% RSLogix 500 project STAR TO DELTA STARTER_BAK003.RSS, saved by version 8.30.00.16 %
PROJECT "UNTITLED"    % processor: Bul.1763 MicroLogix 1100 Series B %

PROGRAM FILES
  LAD 2   4 rungs

DATA FILES
  O0 OUTPUT  4 elements
  I1 INPUT  6 elements
  S2 STATUS  66 elements
  B3 BINARY  1 elements
  T4 TIMER  1 elements
  C5 COUNTER  1 elements
  R6 CONTROL  1 elements
  N7 INTEGER  1 elements
  F8 FLOAT  1 elements

LADDER 2
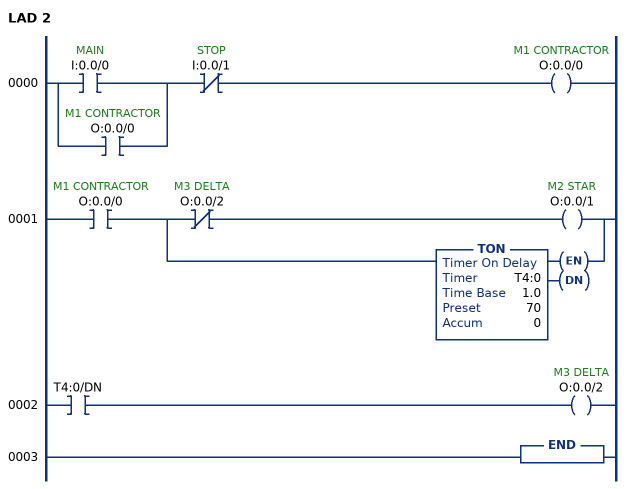
% Rung: 0 %  % edit flag set %
SOR BST XIC I:0.0/0 NXB XIC O:0.0/0 BND XIO I:0.0/1 OTE O:0.0/0 EOR
%   I:0.0/0  "MAIN" %
%   O:0.0/0  "M1 CONTRACTOR" %
%   I:0.0/1  "STOP" %
% Rung: 1 %  % edit flag set %
SOR XIC O:0.0/0 BST XIO O:0.0/2 OTE O:0.0/1 NXB TON T4:0 1.0 70 0 BND EOR
%   O:0.0/0  "M1 CONTRACTOR" %
%   O:0.0/2  "M3 DELTA" %
%   O:0.0/1  "M2 STAR" %
% Rung: 2 %  % edit flag set %
SOR XIC T4:0/DN OTE O:0.0/2 EOR
%   O:0.0/2  "M3 DELTA" %
% Rung: 3 %
SOR END EOR
